ABB RobotStudio station: IRB1600_20220615-165744.rsstn

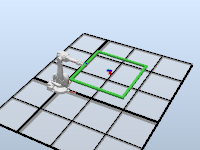
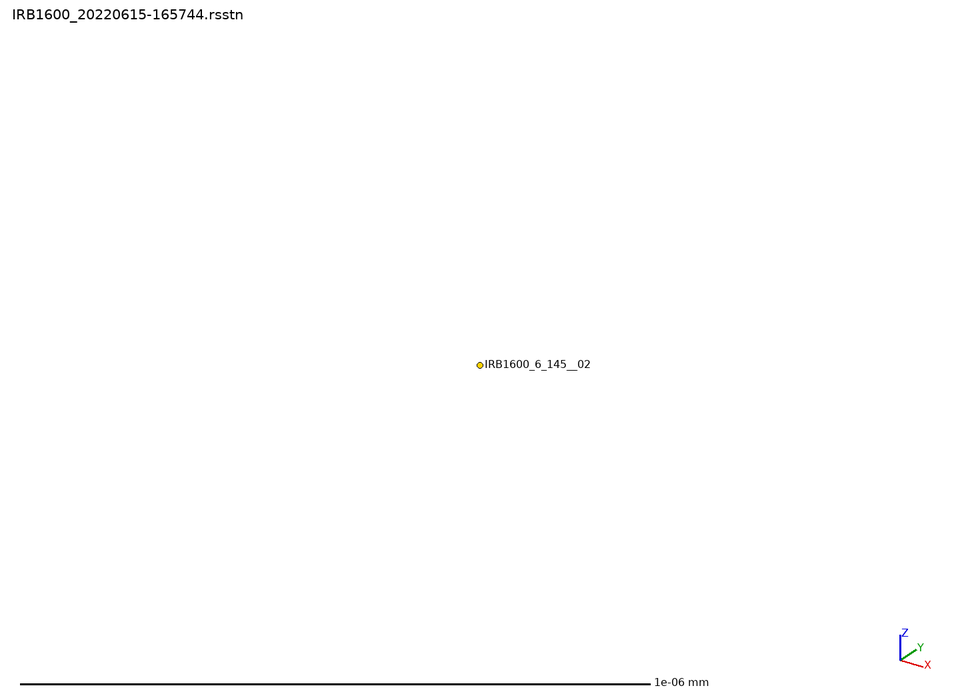
[picture v1: parts stored in the station drawn from their meshes, with robot base, taught points and paths (robot models come from the ABB library and are not in the file)]
Station Solution1 (saved by RobotStudio 22.1.9826.0)
Controller IRB1600_6_145
  mechanical unit ROB_1: IRB1600_6_145__02, 6 joints, base frame (0, 0, 0) mm
Layout (positions relative to the parent item):
  - IRB1600_6_145__02 [mechanism, from Robots\IRB1600_6_145_G_02.rslib] at (0, 0, 0) mm; joint values [-0.0029, -0.0051, 0.0775, -0.04, -0.0725, 0.0399] (rad or m)
  - surface [part] at (1567.14, -2.16, 1115.38) mm, rotated rx 0 ry 0.57 rz 0 deg, size 1500 x 1500 x 50 mm
  - flange_connector [part, from Tools\IsoPlate_small_Binzel.rslib] at (809.88, -2.16, 1143.04) mm, rotated rx 0 ry 90 rz 0 deg
  - Frame_1 [frame] at (1567.14, -2.16, 1115.38) mm, rotated rx 0 ry 0.57 rz 0 deg
Attachment: flange_connector is attached to IRB1600_6_145__02 / Link6
Attachment: Frame_1 is attached to surface
Attachment: surface is attached to flange_connector
Targets, tools, work objects and paths stored in the station, written as RAPID:
! task T_ROB1
MODULE Module1
  LOCAL PERS wobjdata egm_wobj:=[FALSE,TRUE,"",[[0,0,0],[1,0,0,0]],[[0,0,0],[1,0,0,0]]];
  TASK PERS tooldata Tooldata_7:=[TRUE,[[-23.772999698,2.161000196,740.120999999],[0.707106781,0,-0.707106781,0]],[1,[0,0,1],[1,0,0,0],0,0,0]];
  PROC main()
    ConfJ \On;
    MoveJ RelTool (starting_position, 327, 9, 88.8 \Rx:=-17.8, \Ry:=54, \Rz:=0),v400,z1,Tooldata_7;
    MoveJ RelTool (starting_position, 325, 18, 83.3 \Rx:=-17.9, \Ry:=52.5, \Rz:=0),v400,z1,Tooldata_7;
    MoveJ RelTool (starting_position, 322, 27, 77.6 \Rx:=-18, \Ry:=51.3, \Rz:=0),v400,z1,Tooldata_7;
    MoveJ RelTool (starting_position, 319, 27, 71.8 \Rx:=-18.1, \Ry:=49.8, \Rz:=0),v400,z1,Tooldata_7;
    MoveJ RelTool (starting_position, 315, 36, 65.9 \Rx:=-18.1, \Ry:=48.6, \Rz:=0),v400,z1,Tooldata_7;
    MoveJ RelTool (starting_position, 311, 45, 59.4 \Rx:=-18.1, \Ry:=47.7, \Rz:=0),v400,z1,Tooldata_7;
    MoveJ RelTool (starting_position, 307, 54, 52.2 \Rx:=-18.1, \Ry:=46.2, \Rz:=0),v400,z1,Tooldata_7;
    MoveJ RelTool (starting_position, 303, 63, 44.8 \Rx:=-18.1, \Ry:=45, \Rz:=0),v400,z1,Tooldata_7;
    MoveJ RelTool (starting_position, 299, 72, 37.8 \Rx:=-18, \Ry:=44.1, \Rz:=0),v400,z1,Tooldata_7;
    MoveJ RelTool (starting_position, 295, 81, 31.3 \Rx:=-17.8, \Ry:=43.2, \Rz:=0),v400,z1,Tooldata_7;
    MoveJ RelTool (starting_position, 291, 81, 25.2 \Rx:=-17.5, \Ry:=42.3, \Rz:=0),v400,z1,Tooldata_7;
    MoveJ RelTool (starting_position, 287, 90, 18.8 \Rx:=-17.2, \Ry:=41.4, \Rz:=0),v400,z1,Tooldata_7;
    MoveJ RelTool (starting_position, 283, 99, 12.2 \Rx:=-16.7, \Ry:=40.5, \Rz:=0),v400,z1,Tooldata_7;
    MoveJ RelTool (starting_position, 280, 108, 6 \Rx:=-16.2, \Ry:=39.9, \Rz:=0),v400,z1,Tooldata_7;
    MoveJ RelTool (starting_position, 277, 117, 0.1 \Rx:=-15.6, \Ry:=39.6, \Rz:=0),v400,z1,Tooldata_7;
    MoveJ RelTool (starting_position, 275, 126, -6 \Rx:=-15, \Ry:=39, \Rz:=0),v400,z1,Tooldata_7;
    MoveJ RelTool (starting_position, 273, 135, -12.4 \Rx:=-14.1, \Ry:=38.7, \Rz:=0),v400,z1,Tooldata_7;
    MoveJ RelTool (starting_position, 271, 144, -18.5 \Rx:=-13.2, \Ry:=38.4, \Rz:=0),v400,z1,Tooldata_7;
    MoveJ RelTool (starting_position, 269, 153, -24.7 \Rx:=-12.3, \Ry:=38.1, \Rz:=0),v400,z1,Tooldata_7;
    MoveJ RelTool (starting_position, 268, 162, -30.7 \Rx:=-11.3, \Ry:=37.8, \Rz:=0),v400,z1,Tooldata_7;
    MoveJ RelTool (starting_position, 266, 171, -36.7 \Rx:=-10.4, \Ry:=37.5, \Rz:=0),v400,z1,Tooldata_7;
    MoveJ RelTool (starting_position, 265, 180, -42.5 \Rx:=-9.4, \Ry:=37.5, \Rz:=0),v400,z1,Tooldata_7;
    MoveJ RelTool (starting_position, 264, 180, -48 \Rx:=-8.3, \Ry:=37.2, \Rz:=0),v400,z1,Tooldata_7;
    MoveJ RelTool (starting_position, 263, 189, -53.7 \Rx:=-7.4, \Ry:=37.2, \Rz:=0),v400,z1,Tooldata_7;
    MoveJ RelTool (starting_position, 263, 198, -68.8 \Rx:=-6.5, \Ry:=37.2, \Rz:=0),v400,z1,Tooldata_7;
    MoveJ RelTool (starting_position, 262, 207, -82.2 \Rx:=-5.6, \Ry:=36.9, \Rz:=0),v400,z1,Tooldata_7;
    MoveJ RelTool (starting_position, 261, 207, -94.8 \Rx:=-4.9, \Ry:=36.9, \Rz:=0),v400,z1,Tooldata_7;
    MoveJ RelTool (starting_position, 260, 216, -106.8 \Rx:=-4.2, \Ry:=36.6, \Rz:=0),v400,z1,Tooldata_7;
    MoveJ RelTool (starting_position, 259, 225, -118.4 \Rx:=-3.7, \Ry:=36.3, \Rz:=0),v400,z1,Tooldata_7;
    MoveJ RelTool (starting_position, 259, 234, -129.7 \Rx:=-3.3, \Ry:=36, \Rz:=0),v400,z1,Tooldata_7;
    MoveJ RelTool (starting_position, 258, 243, -140.6 \Rx:=-3, \Ry:=36, \Rz:=0),v400,z1,Tooldata_7;
    MoveJ RelTool (starting_position, 257, 252, -151.5 \Rx:=-2.7, \Ry:=36, \Rz:=0),v400,z1,Tooldata_7;
    MoveJ RelTool (starting_position, 257, 261, -162.8 \Rx:=-2.5, \Ry:=36, \Rz:=0),v400,z1,Tooldata_7;
    MoveJ RelTool (starting_position, 256, 261, -174.6 \Rx:=-2.3, \Ry:=35.7, \Rz:=0),v400,z1,Tooldata_7;
    MoveJ RelTool (starting_position, 255, 270, -187 \Rx:=-2.2, \Ry:=35.7, \Rz:=0),v400,z1,Tooldata_7;
    MoveJ RelTool (starting_position, 254, 279, -198.8 \Rx:=-2, \Ry:=35.4, \Rz:=0),v400,z1,Tooldata_7;
    MoveJ RelTool (starting_position, 254, 279, -210.2 \Rx:=-1.8, \Ry:=35.1, \Rz:=0),v400,z1,Tooldata_7;
    MoveJ RelTool (starting_position, 253, 288, -221.7 \Rx:=-1.5, \Ry:=35.1, \Rz:=0),v400,z1,Tooldata_7;
    MoveJ RelTool (starting_position, 252, 297, -233.5 \Rx:=-1.2, \Ry:=34.8, \Rz:=0),v400,z1,Tooldata_7;
    MoveJ RelTool (starting_position, 251, 297, -245.4 \Rx:=-0.9, \Ry:=34.8, \Rz:=0),v400,z1,Tooldata_7;
    MoveJ RelTool (starting_position, 250, 306, -256.8 \Rx:=-0.5, \Ry:=34.5, \Rz:=0),v400,z1,Tooldata_7;
    MoveJ RelTool (starting_position, 249, 315, -267.8 \Rx:=0, \Ry:=34.5, \Rz:=0),v400,z1,Tooldata_7;
    MoveJ RelTool (starting_position, 248, 324, -278.8 \Rx:=0.6, \Ry:=34.2, \Rz:=0),v400,z1,Tooldata_7;
    MoveJ RelTool (starting_position, 247, 333, -290.2 \Rx:=1.1, \Ry:=33.9, \Rz:=0),v400,z1,Tooldata_7;
    MoveJ RelTool (starting_position, 246, 342, -301.6 \Rx:=1.6, \Ry:=33.9, \Rz:=0),v400,z1,Tooldata_7;
    MoveJ RelTool (starting_position, 245, 351, -313.1 \Rx:=2.1, \Ry:=33.6, \Rz:=0),v400,z1,Tooldata_7;
    MoveJ RelTool (starting_position, 243, 351, -324 \Rx:=2.4, \Ry:=33.3, \Rz:=0),v400,z1,Tooldata_7;
    MoveJ RelTool (starting_position, 242, 360, -334.7 \Rx:=2.8, \Ry:=33, \Rz:=0),v400,z1,Tooldata_7;
    MoveJ RelTool (starting_position, 240, 360, -345.4 \Rx:=3.1, \Ry:=32.7, \Rz:=0),v400,z1,Tooldata_7;
    MoveJ RelTool (starting_position, 238, 360, -355.7 \Rx:=3.3, \Ry:=32.4, \Rz:=0),v400,z1,Tooldata_7;
    MoveJ RelTool (starting_position, 236, 360, -365.8 \Rx:=3.4, \Ry:=32.1, \Rz:=0),v400,z1,Tooldata_7;
    MoveJ RelTool (starting_position, 234, 360, -375.5 \Rx:=3.4, \Ry:=31.5, \Rz:=0),v400,z1,Tooldata_7;
    MoveJ RelTool (starting_position, 231, 360, -384.6 \Rx:=3.4, \Ry:=30.9, \Rz:=0),v400,z1,Tooldata_7;
    MoveJ RelTool (starting_position, 228, 369, -393 \Rx:=3.3, \Ry:=30.3, \Rz:=0),v400,z1,Tooldata_7;
    MoveJ RelTool (starting_position, 225, 369, -400.9 \Rx:=3.2, \Ry:=29.7, \Rz:=0),v400,z1,Tooldata_7;
    MoveJ RelTool (starting_position, 221, 378, -408.9 \Rx:=2.9, \Ry:=29.1, \Rz:=0),v400,z1,Tooldata_7;
    MoveJ RelTool (starting_position, 218, 387, -417.2 \Rx:=2.6, \Ry:=28.2, \Rz:=0),v400,z1,Tooldata_7;
    MoveJ RelTool (starting_position, 214, 387, -425.9 \Rx:=2.3, \Ry:=27.3, \Rz:=0),v400,z1,Tooldata_7;
    MoveJ RelTool (starting_position, 210, 396, -433.8 \Rx:=1.9, \Ry:=26.4, \Rz:=0),v400,z1,Tooldata_7;
    MoveJ RelTool (starting_position, 205, 405, -441 \Rx:=1.6, \Ry:=25.5, \Rz:=0),v400,z1,Tooldata_7;
    MoveJ RelTool (starting_position, 201, 414, -448.5 \Rx:=1.2, \Ry:=24.6, \Rz:=0),v400,z1,Tooldata_7;
    MoveJ RelTool (starting_position, 196, 423, -456.4 \Rx:=0.9, \Ry:=23.4, \Rz:=0),v400,z1,Tooldata_7;
    MoveJ RelTool (starting_position, 192, 432, -463.8 \Rx:=0.4, \Ry:=22.5, \Rz:=0),v400,z1,Tooldata_7;
    MoveJ RelTool (starting_position, 187, 441, -470.7 \Rx:=0.1, \Ry:=21.6, \Rz:=0),v400,z1,Tooldata_7;
    MoveJ RelTool (starting_position, 182, 441, -477.9 \Rx:=-0.2, \Ry:=20.4, \Rz:=0),v400,z1,Tooldata_7;
    MoveJ RelTool (starting_position, 178, 450, -485.1 \Rx:=-0.6, \Ry:=19.5, \Rz:=0),v400,z1,Tooldata_7;
    MoveJ RelTool (starting_position, 173, 450, -492.2 \Rx:=-0.8, \Ry:=18.3, \Rz:=0),v400,z1,Tooldata_7;
    MoveJ RelTool (starting_position, 169, 450, -499 \Rx:=-1, \Ry:=17.4, \Rz:=0),v400,z1,Tooldata_7;
    MoveJ RelTool (starting_position, 165, 450, -505.8 \Rx:=-1.1, \Ry:=16.5, \Rz:=0),v400,z1,Tooldata_7;
    MoveJ RelTool (starting_position, 160, 450, -512.6 \Rx:=-1.1, \Ry:=15.6, \Rz:=0),v400,z1,Tooldata_7;
    MoveJ RelTool (starting_position, 157, 450, -519 \Rx:=-1.1, \Ry:=15, \Rz:=0),v400,z1,Tooldata_7;
    MoveJ RelTool (starting_position, 153, 450, -525 \Rx:=-1.1, \Ry:=14.1, \Rz:=0),v400,z1,Tooldata_7;
    MoveJ RelTool (starting_position, 150, 450, -530.7 \Rx:=-1, \Ry:=13.5, \Rz:=0),v400,z1,Tooldata_7;
    MoveJ RelTool (starting_position, 147, 450, -535.9 \Rx:=-0.9, \Ry:=12.9, \Rz:=0),v400,z1,Tooldata_7;
    MoveJ RelTool (starting_position, 144, 450, -540.9 \Rx:=-0.7, \Ry:=12.3, \Rz:=0),v400,z1,Tooldata_7;
    MoveJ RelTool (starting_position, 141, 450, -545.5 \Rx:=-0.6, \Ry:=11.7, \Rz:=0),v400,z1,Tooldata_7;
    MoveJ RelTool (starting_position, 139, 450, -550 \Rx:=-0.4, \Ry:=11.1, \Rz:=0),v400,z1,Tooldata_7;
    MoveJ RelTool (starting_position, 137, 450, -554.5 \Rx:=-0.2, \Ry:=10.8, \Rz:=0),v400,z1,Tooldata_7;
    MoveJ RelTool (starting_position, 135, 450, -559.1 \Rx:=-0.1, \Ry:=10.5, \Rz:=0),v400,z1,Tooldata_7;
    MoveJ RelTool (starting_position, 133, 450, -563.3 \Rx:=-0, \Ry:=10.5, \Rz:=0),v400,z1,Tooldata_7;
    MoveJ RelTool (starting_position, 131, 450, -566.9 \Rx:=0, \Ry:=9.9, \Rz:=0),v400,z1,Tooldata_7;
    MoveJ RelTool (starting_position, 130, 450, -570.1 \Rx:=0, \Ry:=9.6, \Rz:=0),v400,z1,Tooldata_7;
    MoveJ RelTool (starting_position, 128, 450, -573.2 \Rx:=0, \Ry:=9.3, \Rz:=0),v400,z1,Tooldata_7;
    MoveJ RelTool (starting_position, 126, 450, -576.4 \Rx:=-0, \Ry:=9, \Rz:=0),v400,z1,Tooldata_7;
    MoveJ RelTool (starting_position, 125, 450, -579.5 \Rx:=-0.1, \Ry:=9, \Rz:=0),v400,z1,Tooldata_7;
    MoveJ RelTool (starting_position, 123, 450, -582.3 \Rx:=-0.2, \Ry:=8.7, \Rz:=0),v400,z1,Tooldata_7;
    MoveJ RelTool (starting_position, 121, 450, -584.5 \Rx:=-0.3, \Ry:=8.1, \Rz:=0),v400,z1,Tooldata_7;
    MoveJ RelTool (starting_position, 119, 450, -586.8 \Rx:=-0.5, \Ry:=7.8, \Rz:=0),v400,z1,Tooldata_7;
    MoveJ RelTool (starting_position, 117, 450, -589.1 \Rx:=-0.8, \Ry:=7.5, \Rz:=0),v400,z1,Tooldata_7;
    MoveJ RelTool (starting_position, 115, 450, -590.9 \Rx:=-1, \Ry:=6.9, \Rz:=0),v400,z1,Tooldata_7;
    MoveJ RelTool (starting_position, 113, 450, -592.3 \Rx:=-1.3, \Ry:=6.3, \Rz:=0),v400,z1,Tooldata_7;
    MoveJ RelTool (starting_position, 111, 450, -593.3 \Rx:=-1.6, \Ry:=5.7, \Rz:=0),v400,z1,Tooldata_7;
    MoveJ RelTool (starting_position, 108, 450, -594.1 \Rx:=-1.9, \Ry:=5.4, \Rz:=0),v400,z1,Tooldata_7;
    MoveJ RelTool (starting_position, 106, 450, -594.9 \Rx:=-2.1, \Ry:=5.1, \Rz:=0),v400,z1,Tooldata_7;
    MoveJ RelTool (starting_position, 103, 450, -596.1 \Rx:=-2.3, \Ry:=4.5, \Rz:=0),v400,z1,Tooldata_7;
    MoveJ RelTool (starting_position, 100, 450, -597.6 \Rx:=-2.5, \Ry:=3.9, \Rz:=0),v400,z1,Tooldata_7;
    MoveJ RelTool (starting_position, 97, 450, -599.1 \Rx:=-2.7, \Ry:=3.3, \Rz:=0),v400,z1,Tooldata_7;
    MoveJ RelTool (starting_position, 95, 450, -600.2 \Rx:=-2.7, \Ry:=2.7, \Rz:=0),v400,z1,Tooldata_7;
    MoveJ RelTool (starting_position, 92, 450, -600.8 \Rx:=-2.8, \Ry:=1.8, \Rz:=0),v400,z1,Tooldata_7;
    MoveJ RelTool (starting_position, 89, 450, -601.1 \Rx:=-2.8, \Ry:=1.2, \Rz:=0),v400,z1,Tooldata_7;
    MoveJ RelTool (starting_position, 86, 441, -601.1 \Rx:=-2.7, \Ry:=0.6, \Rz:=0),v400,z1,Tooldata_7;
    MoveJ RelTool (starting_position, 83, 441, -601.1 \Rx:=-2.4, \Ry:=0, \Rz:=0),v400,z1,Tooldata_7;
    MoveJ RelTool (starting_position, 80, 432, -601.1 \Rx:=-2.2, \Ry:=-0.3, \Rz:=0),v400,z1,Tooldata_7;
    MoveJ RelTool (starting_position, 77, 423, -600.8 \Rx:=-1.9, \Ry:=-0.9, \Rz:=0),v400,z1,Tooldata_7;
    MoveJ RelTool (starting_position, 74, 423, -600 \Rx:=-1.5, \Ry:=-1.8, \Rz:=0),v400,z1,Tooldata_7;
    MoveJ RelTool (starting_position, 71, 414, -599.6 \Rx:=-1, \Ry:=-2.4, \Rz:=0),v400,z1,Tooldata_7;
    MoveJ RelTool (starting_position, 68, 405, -599.4 \Rx:=-0.4, \Ry:=-3, \Rz:=0),v400,z1,Tooldata_7;
    MoveJ RelTool (starting_position, 64, 396, -599 \Rx:=0.3, \Ry:=-3.6, \Rz:=0),v400,z1,Tooldata_7;
    MoveJ RelTool (starting_position, 61, 387, -597.9 \Rx:=1, \Ry:=-4.2, \Rz:=0),v400,z1,Tooldata_7;
    MoveJ RelTool (starting_position, 58, 378, -596.6 \Rx:=1.7, \Ry:=-5.1, \Rz:=0),v400,z1,Tooldata_7;
    MoveJ RelTool (starting_position, 55, 369, -594.9 \Rx:=2.4, \Ry:=-5.7, \Rz:=0),v400,z1,Tooldata_7;
    MoveJ RelTool (starting_position, 52, 369, -592.4 \Rx:=3.1, \Ry:=-6.3, \Rz:=0),v400,z1,Tooldata_7;
    MoveJ RelTool (starting_position, 49, 360, -590.1 \Rx:=3.9, \Ry:=-6.9, \Rz:=0),v400,z1,Tooldata_7;
    MoveJ RelTool (starting_position, 45, 360, -588.1 \Rx:=4.6, \Ry:=-7.5, \Rz:=0),v400,z1,Tooldata_7;
    MoveJ RelTool (starting_position, 42, 360, -586.1 \Rx:=5.2, \Ry:=-8.4, \Rz:=0),v400,z1,Tooldata_7;
    MoveJ RelTool (starting_position, 39, 360, -583.7 \Rx:=5.8, \Ry:=-9, \Rz:=0),v400,z1,Tooldata_7;
    MoveJ RelTool (starting_position, 36, 360, -580.8 \Rx:=6.3, \Ry:=-9.6, \Rz:=0),v400,z1,Tooldata_7;
    MoveJ RelTool (starting_position, 33, 360, -577.5 \Rx:=6.8, \Ry:=-10.2, \Rz:=0),v400,z1,Tooldata_7;
    MoveJ RelTool (starting_position, 30, 351, -574.3 \Rx:=7.2, \Ry:=-10.8, \Rz:=0),v400,z1,Tooldata_7;
    MoveJ RelTool (starting_position, 28, 351, -571 \Rx:=7.5, \Ry:=-11.4, \Rz:=0),v400,z1,Tooldata_7;
    MoveJ RelTool (starting_position, 25, 342, -567.7 \Rx:=7.6, \Ry:=-12, \Rz:=0),v400,z1,Tooldata_7;
    MoveJ RelTool (starting_position, 22, 333, -564.5 \Rx:=7.6, \Ry:=-12.3, \Rz:=0),v400,z1,Tooldata_7;
    MoveJ RelTool (starting_position, 19, 333, -561.2 \Rx:=7.5, \Ry:=-12.9, \Rz:=0),v400,z1,Tooldata_7;
    MoveJ RelTool (starting_position, 16, 324, -557.9 \Rx:=7.3, \Ry:=-13.5, \Rz:=0),v400,z1,Tooldata_7;
    MoveJ RelTool (starting_position, 13, 315, -554.7 \Rx:=7.1, \Ry:=-14.1, \Rz:=0),v400,z1,Tooldata_7;
    MoveJ RelTool (starting_position, 10, 306, -550.7 \Rx:=6.8, \Ry:=-14.7, \Rz:=0),v400,z1,Tooldata_7;
    MoveJ RelTool (starting_position, 7, 297, -545.9 \Rx:=6.3, \Ry:=-15.3, \Rz:=0),v400,z1,Tooldata_7;
    MoveJ RelTool (starting_position, 4, 288, -540.3 \Rx:=5.9, \Ry:=-15.9, \Rz:=0),v400,z1,Tooldata_7;
    MoveJ RelTool (starting_position, 1, 279, -534.3 \Rx:=5.5, \Ry:=-16.5, \Rz:=0),v400,z1,Tooldata_7;
    MoveJ RelTool (starting_position, -2, 279, -527.6 \Rx:=5.1, \Ry:=-17.1, \Rz:=0),v400,z1,Tooldata_7;
    MoveJ RelTool (starting_position, -6, 270, -520.2 \Rx:=4.7, \Ry:=-18, \Rz:=0),v400,z1,Tooldata_7;
    MoveJ RelTool (starting_position, -9, 261, -511.9 \Rx:=4.4, \Ry:=-18.6, \Rz:=0),v400,z1,Tooldata_7;
    MoveJ RelTool (starting_position, -13, 261, -503 \Rx:=4.3, \Ry:=-19.2, \Rz:=0),v400,z1,Tooldata_7;
    MoveJ RelTool (starting_position, -17, 252, -494 \Rx:=4.2, \Ry:=-20.1, \Rz:=0),v400,z1,Tooldata_7;
    MoveJ RelTool (starting_position, -20, 243, -485 \Rx:=4.3, \Ry:=-21, \Rz:=0),v400,z1,Tooldata_7;
    MoveJ RelTool (starting_position, -24, 243, -475.6 \Rx:=4.5, \Ry:=-21.9, \Rz:=0),v400,z1,Tooldata_7;
    MoveJ RelTool (starting_position, -28, 234, -465.7 \Rx:=4.9, \Ry:=-22.8, \Rz:=0),v400,z1,Tooldata_7;
    MoveJ RelTool (starting_position, -32, 225, -455.8 \Rx:=5.2, \Ry:=-23.7, \Rz:=0),v400,z1,Tooldata_7;
    MoveJ RelTool (starting_position, -35, 216, -447 \Rx:=5.7, \Ry:=-24.6, \Rz:=0),v400,z1,Tooldata_7;
    MoveJ RelTool (starting_position, -39, 207, -438.7 \Rx:=6.2, \Ry:=-25.2, \Rz:=0),v400,z1,Tooldata_7;
    MoveJ RelTool (starting_position, -42, 198, -430.9 \Rx:=6.8, \Ry:=-26.1, \Rz:=0),v400,z1,Tooldata_7;
    MoveJ RelTool (starting_position, -44, 189, -423.3 \Rx:=7.5, \Ry:=-26.7, \Rz:=0),v400,z1,Tooldata_7;
    MoveJ RelTool (starting_position, -46, 180, -416.1 \Rx:=8.2, \Ry:=-27.6, \Rz:=0),v400,z1,Tooldata_7;
    MoveJ RelTool (starting_position, -47, 171, -409.4 \Rx:=8.9, \Ry:=-27.9, \Rz:=0),v400,z1,Tooldata_7;
    MoveJ RelTool (starting_position, -47, 162, -403.6 \Rx:=9.5, \Ry:=-28.2, \Rz:=0),v400,z1,Tooldata_7;
    MoveJ RelTool (starting_position, -47, 162, -398.6 \Rx:=10, \Ry:=-27.9, \Rz:=0),v400,z1,Tooldata_7;
    MoveJ RelTool (starting_position, -45, 153, -394.6 \Rx:=10.3, \Ry:=-27.9, \Rz:=0),v400,z1,Tooldata_7;
    MoveJ RelTool (starting_position, -42, 144, -391.6 \Rx:=10.6, \Ry:=-27.6, \Rz:=0),v400,z1,Tooldata_7;
    MoveJ RelTool (starting_position, -38, 135, -388.2 \Rx:=10.7, \Ry:=-26.7, \Rz:=0),v400,z1,Tooldata_7;
    MoveJ RelTool (starting_position, -32, 126, -384.7 \Rx:=10.6, \Ry:=-25.5, \Rz:=0),v400,z1,Tooldata_7;
    MoveJ RelTool (starting_position, -25, 117, -381.9 \Rx:=10.5, \Ry:=-24.3, \Rz:=0),v400,z1,Tooldata_7;
    MoveJ RelTool (starting_position, -17, 108, -379.6 \Rx:=10.1, \Ry:=-22.5, \Rz:=0),v400,z1,Tooldata_7;
    MoveJ RelTool (starting_position, -8, 99, -377.2 \Rx:=9.6, \Ry:=-20.4, \Rz:=0),v400,z1,Tooldata_7;
    MoveJ RelTool (starting_position, 2, 90, -374.8 \Rx:=9, \Ry:=-18, \Rz:=0),v400,z1,Tooldata_7;
    MoveJ RelTool (starting_position, 14, 81, -372.5 \Rx:=8.3, \Ry:=-15.6, \Rz:=0),v400,z1,Tooldata_7;
    MoveJ RelTool (starting_position, 26, 72, -370.4 \Rx:=7.6, \Ry:=-12.6, \Rz:=0),v400,z1,Tooldata_7;
    MoveJ RelTool (starting_position, 39, 72, -368.7 \Rx:=6.7, \Ry:=-9.6, \Rz:=0),v400,z1,Tooldata_7;
    MoveJ RelTool (starting_position, 53, 63, -367.3 \Rx:=5.8, \Ry:=-6.3, \Rz:=0),v400,z1,Tooldata_7;
    MoveJ RelTool (starting_position, 66, 54, -366.3 \Rx:=4.8, \Ry:=-3, \Rz:=0),v400,z1,Tooldata_7;
    MoveJ RelTool (starting_position, 80, 45, -364.9 \Rx:=3.9, \Ry:=0.3, \Rz:=0),v400,z1,Tooldata_7;
    MoveJ RelTool (starting_position, 94, 27, -363.1 \Rx:=3, \Ry:=3.3, \Rz:=0),v400,z1,Tooldata_7;
    MoveJ RelTool (starting_position, 106, 18, -361.4 \Rx:=2.1, \Ry:=6.3, \Rz:=0),v400,z1,Tooldata_7;
    MoveJ RelTool (starting_position, 119, 9, -360 \Rx:=1.3, \Ry:=9, \Rz:=0),v400,z1,Tooldata_7;
    MoveJ RelTool (starting_position, 130, 9, -359.2 \Rx:=0.5, \Ry:=11.7, \Rz:=0),v400,z1,Tooldata_7;
    MoveJ RelTool (starting_position, 140, -0, -358.7 \Rx:=-0.1, \Ry:=14.1, \Rz:=0),v400,z1,Tooldata_7;
    MoveJ RelTool (starting_position, 149, -9, -358.2 \Rx:=-0.7, \Ry:=16.2, \Rz:=0),v400,z1,Tooldata_7;
    MoveJ RelTool (starting_position, 156, -18, -357.7 \Rx:=-1.1, \Ry:=17.7, \Rz:=0),v400,z1,Tooldata_7;
    MoveJ RelTool (starting_position, 162, -27, -356.9 \Rx:=-1.4, \Ry:=18.9, \Rz:=0),v400,z1,Tooldata_7;
    MoveJ RelTool (starting_position, 167, -36, -355.7 \Rx:=-1.6, \Ry:=19.8, \Rz:=0),v400,z1,Tooldata_7;
    MoveJ RelTool (starting_position, 170, -45, -354.4 \Rx:=-1.7, \Ry:=20.4, \Rz:=0),v400,z1,Tooldata_7;
    MoveJ RelTool (starting_position, 171, -54, -353.6 \Rx:=-1.7, \Ry:=20.4, \Rz:=0),v400,z1,Tooldata_7;
    MoveJ RelTool (starting_position, 171, -63, -353.1 \Rx:=-1.7, \Ry:=20.4, \Rz:=0),v400,z1,Tooldata_7;
    MoveJ RelTool (starting_position, 170, -72, -353.4 \Rx:=-1.5, \Ry:=19.8, \Rz:=0),v400,z1,Tooldata_7;
    MoveJ RelTool (starting_position, 168, -81, -354.5 \Rx:=-1.4, \Ry:=19.2, \Rz:=0),v400,z1,Tooldata_7;
    MoveJ RelTool (starting_position, 165, -90, -356.3 \Rx:=-1.1, \Ry:=18.3, \Rz:=0),v400,z1,Tooldata_7;
    MoveJ RelTool (starting_position, 161, -99, -358.5 \Rx:=-0.8, \Ry:=17.1, \Rz:=0),v400,z1,Tooldata_7;
    MoveJ RelTool (starting_position, 156, -108, -361 \Rx:=-0.5, \Ry:=15.9, \Rz:=0),v400,z1,Tooldata_7;
    MoveJ RelTool (starting_position, 150, -108, -363.8 \Rx:=-0.2, \Ry:=14.7, \Rz:=0),v400,z1,Tooldata_7;
    MoveJ RelTool (starting_position, 144, -117, -367.4 \Rx:=0.2, \Ry:=13.2, \Rz:=0),v400,z1,Tooldata_7;
    MoveJ RelTool (starting_position, 138, -126, -371.8 \Rx:=0.5, \Ry:=11.7, \Rz:=0),v400,z1,Tooldata_7;
    MoveJ RelTool (starting_position, 131, -135, -376.1 \Rx:=0.8, \Ry:=10.2, \Rz:=0),v400,z1,Tooldata_7;
    MoveJ RelTool (starting_position, 124, -144, -380.5 \Rx:=1, \Ry:=8.4, \Rz:=0),v400,z1,Tooldata_7;
    MoveJ RelTool (starting_position, 117, -153, -385.3 \Rx:=1.2, \Ry:=6.9, \Rz:=0),v400,z1,Tooldata_7;
    MoveJ RelTool (starting_position, 110, -162, -390.1 \Rx:=1.3, \Ry:=5.4, \Rz:=0),v400,z1,Tooldata_7;
    MoveJ RelTool (starting_position, 104, -171, -394.4 \Rx:=1.5, \Ry:=3.9, \Rz:=0),v400,z1,Tooldata_7;
    MoveJ RelTool (starting_position, 97, -180, -398.1 \Rx:=1.6, \Ry:=2.7, \Rz:=0),v400,z1,Tooldata_7;
    MoveJ RelTool (starting_position, 91, -189, -401.4 \Rx:=1.8, \Ry:=1.2, \Rz:=0),v400,z1,Tooldata_7;
    MoveJ RelTool (starting_position, 85, -198, -404.3 \Rx:=2.1, \Ry:=0, \Rz:=0),v400,z1,Tooldata_7;
    MoveJ RelTool (starting_position, 79, -198, -406.6 \Rx:=2.3, \Ry:=-1.2, \Rz:=0),v400,z1,Tooldata_7;
    MoveJ RelTool (starting_position, 74, -207, -408.2 \Rx:=2.6, \Ry:=-2.4, \Rz:=0),v400,z1,Tooldata_7;
    MoveJ RelTool (starting_position, 69, -216, -409.2 \Rx:=2.9, \Ry:=-3.3, \Rz:=0),v400,z1,Tooldata_7;
    MoveJ RelTool (starting_position, 64, -225, -409.5 \Rx:=3.2, \Ry:=-4.5, \Rz:=0),v400,z1,Tooldata_7;
    MoveJ RelTool (starting_position, 60, -234, -409.1 \Rx:=3.6, \Ry:=-5.1, \Rz:=0),v400,z1,Tooldata_7;
    MoveJ RelTool (starting_position, 56, -243, -408 \Rx:=4, \Ry:=-5.7, \Rz:=0),v400,z1,Tooldata_7;
    MoveJ RelTool (starting_position, 53, -252, -406.7 \Rx:=4.4, \Ry:=-6.6, \Rz:=0),v400,z1,Tooldata_7;
    MoveJ RelTool (starting_position, 50, -261, -406.3 \Rx:=4.8, \Ry:=-7.2, \Rz:=0),v400,z1,Tooldata_7;
    MoveJ RelTool (starting_position, 47, -261, -405.8 \Rx:=5.3, \Ry:=-7.5, \Rz:=0),v400,z1,Tooldata_7;
    MoveJ RelTool (starting_position, 44, -270, -404.7 \Rx:=5.8, \Ry:=-8.1, \Rz:=0),v400,z1,Tooldata_7;
    MoveJ RelTool (starting_position, 41, -279, -402.8 \Rx:=6.4, \Ry:=-8.7, \Rz:=0),v400,z1,Tooldata_7;
    MoveJ RelTool (starting_position, 39, -279, -400.4 \Rx:=7, \Ry:=-9.3, \Rz:=0),v400,z1,Tooldata_7;
    MoveJ RelTool (starting_position, 36, -288, -398 \Rx:=7.5, \Ry:=-9.6, \Rz:=0),v400,z1,Tooldata_7;
    MoveJ RelTool (starting_position, 34, -297, -395.6 \Rx:=8, \Ry:=-10.2, \Rz:=0),v400,z1,Tooldata_7;
    MoveJ RelTool (starting_position, 32, -297, -393.2 \Rx:=8.5, \Ry:=-10.5, \Rz:=0),v400,z1,Tooldata_7;
    MoveJ RelTool (starting_position, 30, -306, -388.6 \Rx:=8.9, \Ry:=-10.8, \Rz:=0),v400,z1,Tooldata_7;
    MoveJ RelTool (starting_position, 28, -315, -382.7 \Rx:=9.3, \Ry:=-11.1, \Rz:=0),v400,z1,Tooldata_7;
    MoveJ RelTool (starting_position, 27, -324, -376.8 \Rx:=9.7, \Ry:=-11.4, \Rz:=0),v400,z1,Tooldata_7;
    MoveJ RelTool (starting_position, 25, -333, -370.8 \Rx:=10, \Ry:=-11.7, \Rz:=0),v400,z1,Tooldata_7;
    MoveJ RelTool (starting_position, 23, -342, -364.9 \Rx:=10.2, \Ry:=-12.3, \Rz:=0),v400,z1,Tooldata_7;
    MoveJ RelTool (starting_position, 21, -351, -358.7 \Rx:=10.6, \Ry:=-12.6, \Rz:=0),v400,z1,Tooldata_7;
    MoveJ RelTool (starting_position, 19, -351, -351.2 \Rx:=10.9, \Ry:=-12.9, \Rz:=0),v400,z1,Tooldata_7;
    MoveJ RelTool (starting_position, 17, -360, -343.7 \Rx:=11.1, \Ry:=-13.2, \Rz:=0),v400,z1,Tooldata_7;
    MoveJ RelTool (starting_position, 15, -360, -336.2 \Rx:=11.3, \Ry:=-13.5, \Rz:=0),v400,z1,Tooldata_7;
    MoveJ RelTool (starting_position, 13, -360, -328.7 \Rx:=11.5, \Ry:=-13.8, \Rz:=0),v400,z1,Tooldata_7;
    MoveJ RelTool (starting_position, 11, -360, -321.2 \Rx:=11.7, \Ry:=-14.4, \Rz:=0),v400,z1,Tooldata_7;
    MoveJ RelTool (starting_position, 8, -360, -314 \Rx:=11.8, \Ry:=-15, \Rz:=0),v400,z1,Tooldata_7;
    MoveJ RelTool (starting_position, 6, -360, -307.2 \Rx:=11.9, \Ry:=-15.6, \Rz:=0),v400,z1,Tooldata_7;
    MoveJ RelTool (starting_position, 3, -369, -300.1 \Rx:=12, \Ry:=-15.9, \Rz:=0),v400,z1,Tooldata_7;
    MoveJ RelTool (starting_position, 1, -369, -291.6 \Rx:=11.9, \Ry:=-16.5, \Rz:=0),v400,z1,Tooldata_7;
    MoveJ RelTool (starting_position, -2, -378, -283.8 \Rx:=11.8, \Ry:=-17.4, \Rz:=0),v400,z1,Tooldata_7;
    MoveJ RelTool (starting_position, -5, -387, -276.4 \Rx:=11.6, \Ry:=-18, \Rz:=0),v400,z1,Tooldata_7;
    MoveJ RelTool (starting_position, -8, -387, -269 \Rx:=11.3, \Ry:=-18.9, \Rz:=0),v400,z1,Tooldata_7;
    MoveJ RelTool (starting_position, -10, -396, -261.2 \Rx:=11, \Ry:=-19.2, \Rz:=0),v400,z1,Tooldata_7;
    MoveJ RelTool (starting_position, -12, -405, -253.1 \Rx:=10.5, \Ry:=-19.8, \Rz:=0),v400,z1,Tooldata_7;
    MoveJ RelTool (starting_position, -14, -414, -245.4 \Rx:=9.9, \Ry:=-20.4, \Rz:=0),v400,z1,Tooldata_7;
    MoveJ RelTool (starting_position, -16, -423, -238.1 \Rx:=9.2, \Ry:=-20.7, \Rz:=0),v400,z1,Tooldata_7;
    MoveJ RelTool (starting_position, -17, -432, -230.9 \Rx:=8.5, \Ry:=-21.3, \Rz:=0),v400,z1,Tooldata_7;
    MoveJ RelTool (starting_position, -18, -441, -223.3 \Rx:=7.8, \Ry:=-21.6, \Rz:=0),v400,z1,Tooldata_7;
    MoveJ RelTool (starting_position, -19, -441, -214.4 \Rx:=7, \Ry:=-21.6, \Rz:=0),v400,z1,Tooldata_7;
    MoveJ RelTool (starting_position, -19, -450, -205.6 \Rx:=6.2, \Ry:=-21.6, \Rz:=0),v400,z1,Tooldata_7;
    MoveJ RelTool (starting_position, -19, -450, -196.7 \Rx:=5.4, \Ry:=-21.6, \Rz:=0),v400,z1,Tooldata_7;
    MoveJ RelTool (starting_position, -18, -450, -188.3 \Rx:=4.6, \Ry:=-21, \Rz:=0),v400,z1,Tooldata_7;
    MoveJ RelTool (starting_position, -17, -450, -180.6 \Rx:=3.8, \Ry:=-20.7, \Rz:=0),v400,z1,Tooldata_7;
    MoveJ RelTool (starting_position, -15, -450, -174 \Rx:=3.1, \Ry:=-20.4, \Rz:=0),v400,z1,Tooldata_7;
    MoveJ RelTool (starting_position, -13, -450, -167.3 \Rx:=2.3, \Ry:=-20.1, \Rz:=0),v400,z1,Tooldata_7;
    MoveJ RelTool (starting_position, -11, -450, -159.6 \Rx:=1.6, \Ry:=-19.5, \Rz:=0),v400,z1,Tooldata_7;
    MoveJ RelTool (starting_position, -9, -450, -151.7 \Rx:=0.9, \Ry:=-18.9, \Rz:=0),v400,z1,Tooldata_7;
    MoveJ RelTool (starting_position, -6, -450, -143.7 \Rx:=0.3, \Ry:=-18.3, \Rz:=0),v400,z1,Tooldata_7;
    MoveJ RelTool (starting_position, -4, -450, -135.7 \Rx:=-0.2, \Ry:=-17.7, \Rz:=0),v400,z1,Tooldata_7;
    MoveJ RelTool (starting_position, -1, -450, -131.2 \Rx:=-0.7, \Ry:=-17.1, \Rz:=0),v400,z1,Tooldata_7;
    MoveJ RelTool (starting_position, 1, -450, -126.9 \Rx:=-1.1, \Ry:=-16.5, \Rz:=0),v400,z1,Tooldata_7;
    MoveJ RelTool (starting_position, 4, -450, -122.3 \Rx:=-1.5, \Ry:=-15.9, \Rz:=0),v400,z1,Tooldata_7;
    MoveJ RelTool (starting_position, 6, -450, -117.1 \Rx:=-1.8, \Ry:=-15.3, \Rz:=0),v400,z1,Tooldata_7;
    MoveJ RelTool (starting_position, 9, -450, -111.1 \Rx:=-1.9, \Ry:=-15, \Rz:=0),v400,z1,Tooldata_7;
    MoveJ RelTool (starting_position, 11, -450, -104.8 \Rx:=-2, \Ry:=-14.4, \Rz:=0),v400,z1,Tooldata_7;
    MoveJ RelTool (starting_position, 14, -450, -98.2 \Rx:=-2.1, \Ry:=-14.1, \Rz:=0),v400,z1,Tooldata_7;
    MoveJ RelTool (starting_position, 16, -450, -91.8 \Rx:=-2, \Ry:=-13.5, \Rz:=0),v400,z1,Tooldata_7;
    MoveJ RelTool (starting_position, 18, -450, -85.6 \Rx:=-1.9, \Ry:=-12.9, \Rz:=0),v400,z1,Tooldata_7;
    MoveJ RelTool (starting_position, 20, -450, -79.1 \Rx:=-1.8, \Ry:=-12.6, \Rz:=0),v400,z1,Tooldata_7;
    MoveJ RelTool (starting_position, 22, -450, -72.2 \Rx:=-1.6, \Ry:=-12.3, \Rz:=0),v400,z1,Tooldata_7;
    MoveJ RelTool (starting_position, 23, -450, -65 \Rx:=-1.4, \Ry:=-12, \Rz:=0),v400,z1,Tooldata_7;
    MoveJ RelTool (starting_position, 25, -450, -60.3 \Rx:=-1.1, \Ry:=-11.7, \Rz:=0),v400,z1,Tooldata_7;
    MoveJ RelTool (starting_position, 26, -450, -57.2 \Rx:=-0.8, \Ry:=-11.1, \Rz:=0),v400,z1,Tooldata_7;
    MoveJ RelTool (starting_position, 28, -450, -54 \Rx:=-0.5, \Ry:=-10.8, \Rz:=0),v400,z1,Tooldata_7;
    MoveJ RelTool (starting_position, 29, -450, -50.5 \Rx:=-0.2, \Ry:=-10.8, \Rz:=0),v400,z1,Tooldata_7;
    MoveJ RelTool (starting_position, 30, -450, -46.7 \Rx:=0, \Ry:=-10.5, \Rz:=0),v400,z1,Tooldata_7;
    MoveJ RelTool (starting_position, 31, -450, -43.3 \Rx:=0.2, \Ry:=-10.5, \Rz:=0),v400,z1,Tooldata_7;
    MoveJ RelTool (starting_position, 32, -450, -41.7 \Rx:=0.5, \Ry:=-10.2, \Rz:=0),v400,z1,Tooldata_7;
    MoveJ RelTool (starting_position, 32, -450, -40.1 \Rx:=0.7, \Ry:=-9.9, \Rz:=0),v400,z1,Tooldata_7;
    MoveJ RelTool (starting_position, 33, -450, -38.3 \Rx:=0.9, \Ry:=-9.9, \Rz:=0),v400,z1,Tooldata_7;
    MoveJ RelTool (starting_position, 33, -450, -36.3 \Rx:=1.1, \Ry:=-9.6, \Rz:=0),v400,z1,Tooldata_7;
    MoveJ RelTool (starting_position, 34, -450, -34.2 \Rx:=1.3, \Ry:=-9.6, \Rz:=0),v400,z1,Tooldata_7;
  ENDPROC
  PROC EGM_CARTESIAN_MOVE()
    WaitTime 2;
  ENDPROC
  PROC RAPID_MOVE()
  ENDPROC
ENDMODULE

! task T_ROB1
MODULE CalibData
  TASK PERS tooldata Tooldata_4:=[TRUE,[[0,0,0],[1,0,0,0]],[1,[0,0,1],[1,0,0,0],0,0,0]];
  TASK PERS tooldata Tooldata_5:=[TRUE,[[0,0,0],[1,0,0,0]],[1,[0,0,1],[1,0,0,0],0,0,0]];
  TASK PERS tooldata Tooldata_6:=[TRUE,[[0,0,0],[1,0,0,0]],[1,[0,0,1],[1,0,0,0],0,0,0]];
ENDMODULE

